// TIA Portal V20 export
TYPE "LER_typeCommunicationDataR2S"
// stored: Access Published
   STRUCT
      UnitStatus { S7_SetPoint := 'True'} : "LER_typeCommunicationUnitStatus";
      PartData { S7_SetPoint := 'True'} : "LER_typePartDataReelCut";
      PDR { S7_SetPoint := 'True'} : "LER_typePDR";
      InterfaceData { S7_SetPoint := 'True'} : "LER_typeCommunicationInterfaceData";
   END_STRUCT;
END_TYPE
